// TIA Portal project "Pozitif-Negatif Kenar Tetikleme Uygulaması" (V18)

(* hardware
DEVICE "S7-1200 station_1"  S7-1200 Station
   slot 0: "Rack_0"  S7-1200 Rack  Rack  V1.0
   slot 1: "PLC_1"  CPU 1214C AC/DC/Rly  6ES7 214-1BG40-0XB0  V4.6
*)

// ===== PLC "PLC_1"  CPU 1214C AC/DC/Rly =====

VAR_GLOBAL   // PLC tag table "Default tag table"
   "Stop" AT %I0.0 : Bool;
   "PKT" AT %I0.1 : Bool;
   "NKT" AT %I0.2 : Bool;
   "PKT_Yardımcı" AT %M0.0 : Bool;
   "Motor_1" AT %Q0.0 : Bool;
   "NKT_Yardımcı" AT %M0.1 : Bool;
   "Motor_2" AT %Q0.1 : Bool;
END_VAR

ORGANIZATION_BLOCK "Main"   // OB1, LAD, ProgramCycle
TITLE = "Main Program Sweep (Cycle)"
{ S7_Optimized_Access := 'TRUE' }
VERSION : 0.1
   VAR_INPUT
      Initial_Call : Bool;   // Initial call of this OB
      Remanence : Bool;   // =True, if remanent data are available
   END_VAR
   VAR_TEMP   // added for the SCL form of the ladder/FBD networks
      _w1 : Bool;
   END_VAR
BEGIN

REGION Network 1
   // Pozitif  Kenar Tetikleme butona bastığım anda sadece 1 döngülük çıkış verir.
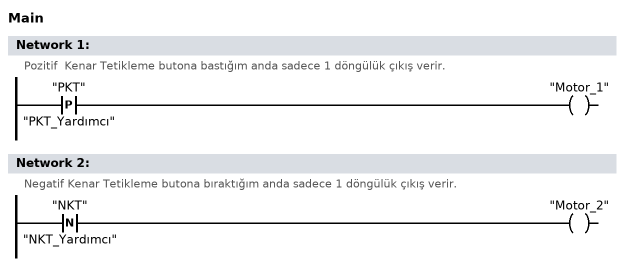
   RUNG wire#powerrail
      P_Contact(operand := "PKT", bit := "PKT_Yardımcı")
      Coil( "Motor_1" )
   END_RUNG
   // the same network as SCL:
   #_w1 := "PKT" AND NOT "PKT_Yardımcı";   // rising edge of "PKT"
   "PKT_Yardımcı" := "PKT";
   "Motor_1" := #_w1;
END_REGION

REGION Network 2
   // Negatif Kenar Tetikleme butona bıraktığım anda sadece 1 döngülük çıkış verir.
   RUNG wire#powerrail
      N_Contact(operand := "NKT", bit := "NKT_Yardımcı")
      Coil( "Motor_2" )
   END_RUNG
   // the same network as SCL:
   #_w1 := NOT "NKT" AND "NKT_Yardımcı";   // falling edge of "NKT"
   "NKT_Yardımcı" := "NKT";
   "Motor_2" := #_w1;
END_REGION
END_ORGANIZATION_BLOCK